ABB RAPID module: Wobj_rfl_locexp_mdfplate.mod

MODULE Wobj_rfl_locexp_mdfplate
	! Points are read in order of declaration.
  ! Please do not change the order of points!

  LOCAL PERS robtarget pWobj_U_PointX1:=[[1797.042,-474.7809,-520.8755],[0.349422752857208,0.680935084819794,0.631367743015289,-0.124923557043076],[0,-2,2,0],[9E+09,9E+09,9E+09,9E+09,9E+09,9E+09]];
	LOCAL PERS robtarget pWobj_U_PointX2:=[[1799.122,-474.1699,387.1608],[0.349396884441376,0.680940091609955,0.631373643875122,-0.124938860535622],[0,-1,1,0],[9E+09,9E+09,9E+09,9E+09,9E+09,9E+09]];
	LOCAL PERS robtarget pWobj_U_PointY1:=[[1718.109,-1079.292,387.1527],[0.418926239013672,0.64184296131134,0.638848185539246,-0.0664184838533401],[-1,-1,1,0],[9E+09,9E+09,9E+09,9E+09,9E+09,9E+09]];

ENDMODULE
